FUNCTION_BLOCK DoorMove (* Basic Function Block Type *)
  (* Standard: 61499-2 *)
  (* Version 0.0, 6/3/2016, Andrei, nxtControl GmbH, Template *)
  PACKAGE Main;
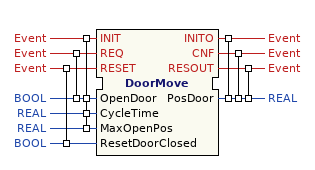
  EVENT_INPUT
    INIT WITH OpenDoor, CycleTime, MaxOpenPos; (* Initialization Request *)
    REQ WITH OpenDoor; (* Normal Execution Request *)
    RESET WITH ResetDoorClosed;
  END_EVENT
  EVENT_OUTPUT
    INITO WITH PosDoor; (* Initialization Confirm *)
    CNF WITH PosDoor; (* Execution Confirmation *)
    RESOUT WITH PosDoor;
  END_EVENT
  VAR_INPUT
    OpenDoor : BOOL; (* Input event qualifier *)
    CycleTime : REAL;
    MaxOpenPos : REAL;
    ResetDoorClosed : BOOL;
  END_VAR
  VAR_OUTPUT
    PosDoor : REAL; (* Output event qualifier *)
  END_VAR
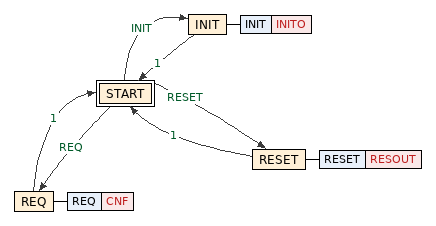
  EC_STATES
    START; (* Initial State *)
    INIT : INIT -> INITO; (* Initialization *)
    REQ : REQ -> CNF; (* Normal execution *)
    RESET : RESET -> RESOUT;
  END_STATES
  EC_TRANSITIONS
    START TO INIT := INIT;
    INIT TO START := 1;
    START TO REQ := REQ;
    REQ TO START := 1;
    START TO RESET := RESET;
    RESET TO START := 1;
  END_TRANSITIONS
  ALGORITHM INIT IN ST: (* Initialization algorithm *)
PosDoor := 0.0;
  END_ALGORITHM
  ALGORITHM REQ IN ST: (* Normally executed algorithm *)
(*IF OpenDoor AND (PosDoor + 50*CycleTime < MaxOpenPos) THEN
	PosDoor := PosDoor + 50 * CycleTime;
ELSIF OpenDoor AND (PosDoor + 50*CycleTime > MaxOpenPos) THEN
	PosDoor := MaxOpenPos;
ELSIF NOT(OpenDoor) AND (PosDoor - 50*CycleTime > 0.0) THEN
	PosDoor := PosDoor - 50 * CycleTime;
ELSIF NOT(OpenDoor) AND (PosDoor - 50*CycleTime < 0.0) THEN
	PosDoor := 0.0;
ELSE
	PosDoor := PosDoor;
END_IF;*)
IF OpenDoor AND (PosDoor < MaxOpenPos) THEN
	PosDoor := MaxOpenPos;
ELSIF OpenDoor AND (PosDoor > MaxOpenPos) THEN
	PosDoor := MaxOpenPos;
ELSIF NOT(OpenDoor) AND (PosDoor > 0.0) THEN
	PosDoor := 0;
ELSIF NOT(OpenDoor) AND (PosDoor < 0.0) THEN
	PosDoor := 0.0;
ELSE
	PosDoor := PosDoor;
END_IF;

(*IF OpenDoor AND (PosDoor < MaxOpenPos) THEN
	PosDoor := -1;
ELSIF OpenDoor AND (PosDoor > MaxOpenPos) THEN
	PosDoor := -1;
ELSIF NOT(OpenDoor) AND (PosDoor > 0.0) THEN
	PosDoor := -1;
ELSIF NOT(OpenDoor) AND (PosDoor < 0.0) THEN
	PosDoor := -1;
ELSE
	PosDoor := -1;
END_IF;*)
  END_ALGORITHM
  ALGORITHM RESET IN ST:
IF (ResetDoorClosed) THEN
	PosDoor := 0.0;
ELSE
	PosDoor := MaxOpenPos;
END_IF;
  END_ALGORITHM
END_FUNCTION_BLOCK
